(* IEC 61131-3 sources: OpenPLC-Project/Code/Blink/build, 1 file *)

(* ---- plc.st ---- *)
TYPE
  LOGLEVEL : (CRITICAL, WARNING, INFO, DEBUG) := INFO;
END_TYPE

FUNCTION_BLOCK LOGGER
  VAR_INPUT
    TRIG : BOOL;
    MSG : STRING;
    LEVEL : LOGLEVEL := INFO;
  END_VAR
  VAR
    TRIG0 : BOOL;
  END_VAR

  IF TRIG AND NOT TRIG0 THEN
  {{
   LogMessage(GetFbVar(LEVEL),(char*)GetFbVar(MSG, .body),GetFbVar(MSG, .len));
  }}
  END_IF;
  TRIG0:=TRIG;
END_FUNCTION_BLOCK

PROGRAM Blink
  VAR
    blink_led AT %QX0.0 : BOOL;
  END_VAR
  VAR
    TON0 : TON;
    TOF0 : TOF;
  END_VAR

  TON0(EN := TRUE, IN := NOT(blink_led), PT := T#500ms);
  TOF0(EN := TON0.ENO, IN := TON0.Q, PT := T#500ms);
  blink_led := TOF0.Q;
END_PROGRAM

CONFIGURATION Config0

  RESOURCE Res0 ON PLC
    TASK task0(INTERVAL := T#20ms,PRIORITY := 0);
    PROGRAM instance0 WITH task0 : Blink;
  END_RESOURCE
END_CONFIGURATION
